Omron Sysmac Studio project comunicacion de PLC (Sysmac Studio 1.23.0.14, StandardProject)

# Controller NX1_2: NX1P2-1040DT1 version 1.18
Task PrimaryTask (priority 4, period or condition 2000): Programa0

VAR_GLOBAL
    HMI_CAMBIO_MOTORES AT %W1.0 : BOOL;  (* published *)
    HMI_MOTOR_ENCENDIDO AT %W1.2 : BOOL;  (* published *)
    hmi_pulsador_marcha1 AT %W0.00 : BOOL;  (* published *)
    hmi_pulsador_paro1 AT %W0.02 : BOOL;  (* published *)
    hmi_pulsador_inversion1 AT %W0.04 : BOOL;  (* published *)
    adelante : BOOL;  (* at BuiltInIO://cpu/#0/Output_Bit_00; network input *)
    hmi_velocidades_motor1 AT %W0.14 : BOOL;  (* published *)
    hmi_velocidades_motor2 AT %W0.12 : BOOL;  (* published *)
END_VAR
VAR_GLOBAL RETAIN
    hz_motor1_hmi AT %D6 : INT;  (* published *)
    hz_motor2_hmi AT %D4 : INT;  (* published *)
END_VAR
VAR_GLOBAL
    velocidades_motor1 : BOOL;  (* network output *)
    velocidades_motor2 : BOOL;  (* network input *)
    hz_motor1_envio : INT;  (* network input *)
    hz_motor2_envio : INT;  (* network output *)
    atras : BOOL;  (* at BuiltInIO://cpu/#0/Output_Bit_01 *)
    v1 : BOOL;  (* at BuiltInIO://cpu/#0/Output_Bit_02 *)
    v2 : BOOL;  (* at BuiltInIO://cpu/#0/Output_Bit_03 *)
    pulsador_marcha2 AT %W0.06 : BOOL;  (* published *)
    pulsador_paro2 AT %W0.08 : BOOL;  (* published *)
    pulsador_inversion2 AT %W0.10 : BOOL;  (* published *)
    NX1_2_PM_HMI_MOTOR2 : BOOL;  (* network input *)
    NX1_2_PP_HMI_MOTOR2 : BOOL;  (* network input *)
    NX1_2_INVERTIR_HMI_MOTOR2 : BOOL;  (* network input *)
    NX1_2_MOTOR2_ADELANTE : BOOL;  (* network input *)
    NX1_2_MOTOR2_ATRAS : BOOL;  (* network input *)
    NX1_2_PM_HMI_MOTOR1 : BOOL;  (* network output *)
    NX1_2_PP_HMI_MOTOR1 : BOOL;  (* network output *)
    NX1_2_INVERTIR_HMI_MOTOR1 : BOOL;  (* network output *)
    NX1_2_MOTOR1_ADELANTE : BOOL;  (* network output *)
    NX1_2_MOTOR1_ATRAS : BOOL;  (* network output *)
    marcha2 : BOOL;  (* at BuiltInIO://cpu/#0/Input_Bit_00 *)
    paro2 : BOOL;  (* at BuiltInIO://cpu/#0/Input_Bit_01 *)
    invertir2 : BOOL;  (* at BuiltInIO://cpu/#0/Input_Bit_02 *)
END_VAR

PROGRAM Programa0
VAR
    velocidadmotor2 : INT;
    sentido_telerruptor : BOOL;
    variableinversion : BOOL;
    PARO_BOTONERA : BOOL;
    PARO : BOOL;
END_VAR
VAR_EXTERNAL
    adelante : BOOL;
    atras : BOOL;
    hmi_pulsador_marcha1 : BOOL;
    NX1_2_PM_HMI_MOTOR2 : BOOL;
    hmi_pulsador_paro1 : BOOL;
    NX1_2_PP_HMI_MOTOR2 : BOOL;
    hmi_pulsador_inversion1 : BOOL;
    NX1_2_INVERTIR_HMI_MOTOR2 : BOOL;
    v1 : BOOL;
    v2 : BOOL;
    hmi_velocidades_motor2 : BOOL;
    velocidades_motor1 : BOOL;
    hmi_velocidades_motor1 : BOOL;
    velocidades_motor2 : BOOL;
    pulsador_marcha2 : BOOL;
    NX1_2_PM_HMI_MOTOR1 : BOOL;
    pulsador_paro2 : BOOL;
    NX1_2_PP_HMI_MOTOR1 : BOOL;
    NX1_2_INVERTIR_HMI_MOTOR1 : BOOL;
    pulsador_inversion2 : BOOL;
    hz_motor2_envio : INT;
    hz_motor1_envio : INT;
    hz_motor2_hmi : INT;
    hz_motor1_hmi : INT;
    invertir2 : BOOL;
    marcha2 : BOOL;
    paro2 : BOOL;
    HMI_CAMBIO_MOTORES : BOOL;
    HMI_MOTOR_ENCENDIDO : BOOL;
END_VAR
VAR
    _p1 : BOOL;
    _e2 : R_TRIG;
    _e3 : R_TRIG;
    _e4 : R_TRIG;
END_VAR

(* Section Sección0: ladder, written here as Structured Text *)

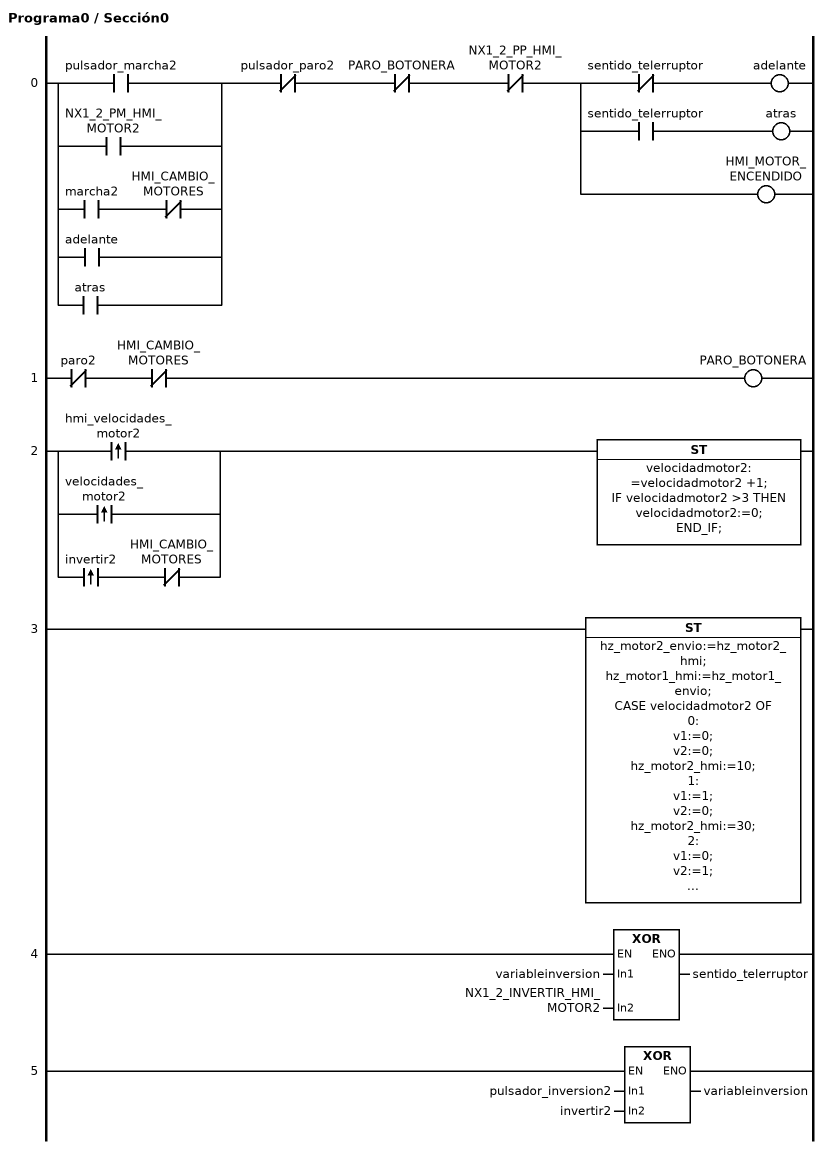
(* Rung 0 *)
_p1 := (pulsador_marcha2 OR NX1_2_PM_HMI_MOTOR2 OR (marcha2 AND NOT HMI_CAMBIO_MOTORES) OR adelante OR atras) AND NOT pulsador_paro2 AND NOT PARO_BOTONERA AND NOT NX1_2_PP_HMI_MOTOR2;
adelante := _p1 AND NOT sentido_telerruptor;
atras := _p1 AND sentido_telerruptor;
HMI_MOTOR_ENCENDIDO := _p1;
(* Rung 1 *)
PARO_BOTONERA := NOT paro2 AND NOT HMI_CAMBIO_MOTORES;
(* Rung 2 *)
_e2(CLK := hmi_velocidades_motor2);
_e3(CLK := velocidades_motor2);
_e4(CLK := invertir2);
IF _e2.Q OR _e3.Q OR (_e4.Q AND NOT HMI_CAMBIO_MOTORES) THEN
    velocidadmotor2:=velocidadmotor2 +1;
    IF velocidadmotor2 >3 THEN
    	velocidadmotor2:=0;
    END_IF;
END_IF;
(* Rung 3 *)
hz_motor2_envio:=hz_motor2_hmi;

hz_motor1_hmi:=hz_motor1_envio;

CASE velocidadmotor2 OF 
	0:
	v1:=0;
	v2:=0;
	hz_motor2_hmi:=10;
	1:
	v1:=1;
	v2:=0;
	hz_motor2_hmi:=30;
	2:
	v1:=0;
	v2:=1;
	hz_motor2_hmi:=50;
	3:
	v1:=1;
	v2:=1;
	hz_motor2_hmi:=80;
END_CASE;



	
(* Rung 4 *)
sentido_telerruptor := variableinversion XOR NX1_2_INVERTIR_HMI_MOTOR2;
(* Rung 5 *)
variableinversion := pulsador_inversion2 XOR invertir2;

(* Section Sección1: ladder, written here as Structured Text *)

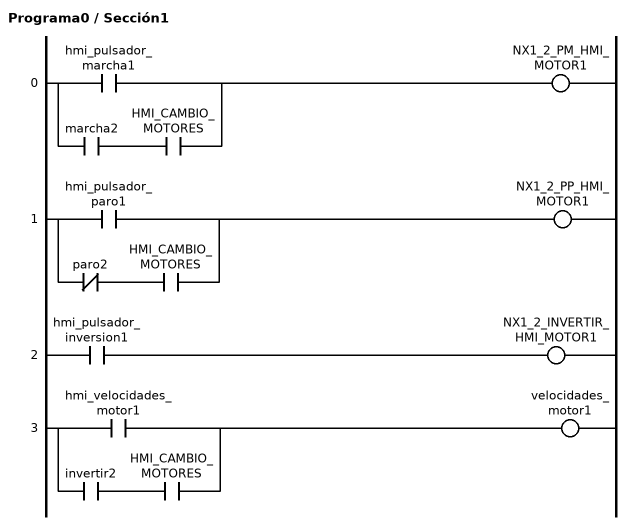
(* Rung 0 *)
NX1_2_PM_HMI_MOTOR1 := hmi_pulsador_marcha1 OR (marcha2 AND HMI_CAMBIO_MOTORES);
(* Rung 1 *)
NX1_2_PP_HMI_MOTOR1 := hmi_pulsador_paro1 OR (NOT paro2 AND HMI_CAMBIO_MOTORES);
(* Rung 2 *)
NX1_2_INVERTIR_HMI_MOTOR1 := hmi_pulsador_inversion1;
(* Rung 3 *)
velocidades_motor1 := hmi_velocidades_motor1 OR (invertir2 AND HMI_CAMBIO_MOTORES);
END_PROGRAM

# Controller NX1_1: NX1P2-1040DT1 version 1.18
Task PrimaryTask (priority 4, period or condition 2000): Programa0

VAR_GLOBAL
    NX1_1_Velocidades_Motor2 : BOOL;  (* network output *)
    NX1_1_Velocidades_Motor1 : BOOL;  (* network input *)
    Velocidades_Motor2_HMI AT %W0.12 : BOOL;  (* published *)
    Velocidades_Motor1_HMI AT %W0.14 : BOOL;  (* published *)
END_VAR
VAR_GLOBAL RETAIN
    Hz_Motor2_HMI AT %D2 : INT;  (* published *)
    Hz_Motor1_HMI AT %D6 : INT;  (* published *)
END_VAR
VAR_GLOBAL
    NX1_1_Hz_Motor2 : INT;  (* network input *)
    NX1_1_Hz_Motor1 : INT;  (* network output *)
    PM1_HMI AT %W0.00 : BOOL;  (* published *)
    PP1_HMI AT %W0.02 : BOOL;  (* published *)
    Invertir1_HMI AT %W0.04 : BOOL;  (* published *)
    PM2_HMI AT %W0.06 : BOOL;  (* published *)
    PP2_HMI AT %W0.08 : BOOL;  (* published *)
    Invertir2_HMI AT %W0.10 : BOOL;  (* published *)
    Motor_Adelante : BOOL;  (* at BuiltInIO://cpu/#0/Output_Bit_00 *)
    Motor_Atras : BOOL;  (* at BuiltInIO://cpu/#0/Output_Bit_01 *)
    NX1_1_PM_HMI_Motor1 : BOOL;  (* network input *)
    NX1_1_PP_HMI_Motor1 : BOOL;  (* network input *)
    NX1_1_Invertir_HMI_Motor1 : BOOL;  (* network input *)
    NX1_1_Motor1_Adelante : BOOL;  (* network input *)
    NX1_1_Motor1_Atras : BOOL;  (* network input *)
    NX1_1_PM_HMI_Motor2 : BOOL;  (* network output *)
    NX1_1_PP_HMI_Motor2 : BOOL;  (* network output *)
    NX1_1_Invertir_HMI_Motor2 : BOOL;  (* network output *)
    NX1_1_Motor2_Adelante : BOOL;  (* network output *)
    NX1_1_Motor2_Atras : BOOL;  (* network output *)
    MV1 : BOOL;  (* at BuiltInIO://cpu/#0/Output_Bit_02 *)
    MV2 : BOOL;  (* at BuiltInIO://cpu/#0/Output_Bit_03 *)
END_VAR

PROGRAM Programa0
VAR
    Sentido : BOOL;
    Velocidad_Motor1 : INT;
END_VAR
VAR_EXTERNAL
    Motor_Adelante : BOOL;
    Motor_Atras : BOOL;
    NX1_1_PM_HMI_Motor1 : BOOL;
    NX1_1_Motor1_Adelante : BOOL;
    NX1_1_Motor1_Atras : BOOL;
    NX1_1_Invertir_HMI_Motor1 : BOOL;
    NX1_1_PP_HMI_Motor1 : BOOL;
    PM1_HMI : BOOL;
    Invertir1_HMI : BOOL;
    PP1_HMI : BOOL;
    PM2_HMI : BOOL;
    NX1_1_Motor2_Adelante : BOOL;
    NX1_1_Motor2_Atras : BOOL;
    PP2_HMI : BOOL;
    Invertir2_HMI : BOOL;
    NX1_1_PM_HMI_Motor2 : BOOL;
    NX1_1_PP_HMI_Motor2 : BOOL;
    NX1_1_Invertir_HMI_Motor2 : BOOL;
    Velocidades_Motor1_HMI : BOOL;
    MV1 : BOOL;
    MV2 : BOOL;
    Velocidades_Motor2_HMI : BOOL;
    NX1_1_Velocidades_Motor1 : BOOL;
    NX1_1_Velocidades_Motor2 : BOOL;
    Hz_Motor1_HMI : INT;
    NX1_1_Hz_Motor1 : INT;
    NX1_1_Hz_Motor2 : INT;
    Hz_Motor2_HMI : INT;
END_VAR
VAR
    _p1 : BOOL;
    _e2 : R_TRIG;
    _e3 : R_TRIG;
END_VAR

(* Section Sección0: ladder, written here as Structured Text *)

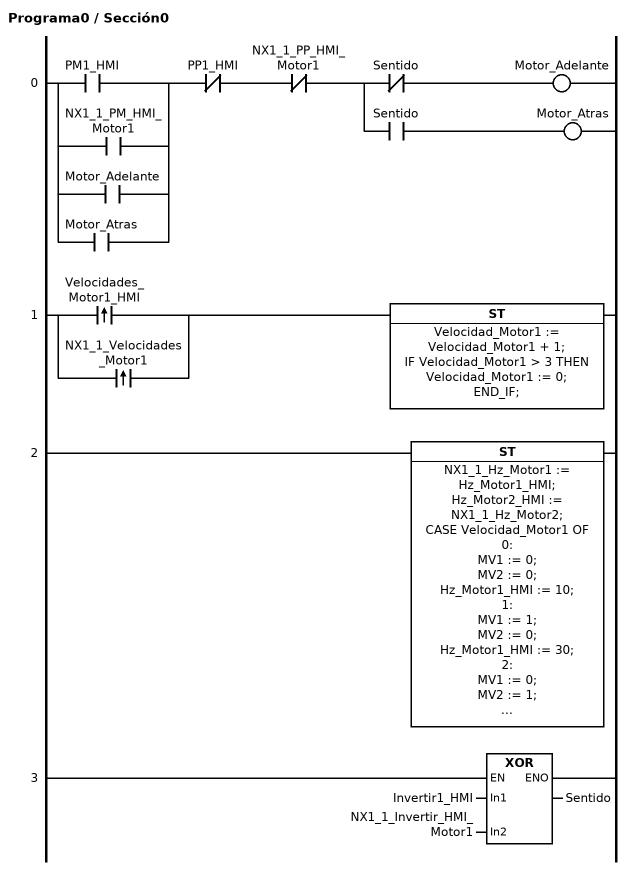
(* Rung 0 *)
_p1 := (PM1_HMI OR NX1_1_PM_HMI_Motor1 OR Motor_Adelante OR Motor_Atras) AND NOT PP1_HMI AND NOT NX1_1_PP_HMI_Motor1;
Motor_Adelante := _p1 AND NOT Sentido;
Motor_Atras := _p1 AND Sentido;
(* Rung 1 *)
_e2(CLK := Velocidades_Motor1_HMI);
_e3(CLK := NX1_1_Velocidades_Motor1);
IF _e2.Q OR _e3.Q THEN
    Velocidad_Motor1 := Velocidad_Motor1 + 1;
    IF Velocidad_Motor1 > 3 THEN
    	Velocidad_Motor1 := 0;
    END_IF;
END_IF;
(* Rung 2 *)
NX1_1_Hz_Motor1 := Hz_Motor1_HMI;
Hz_Motor2_HMI := NX1_1_Hz_Motor2;

CASE Velocidad_Motor1 OF
    0:
	MV1 := 0;
	MV2 := 0;
	Hz_Motor1_HMI := 10;
	1:
	MV1 := 1;
	MV2 := 0;
	Hz_Motor1_HMI := 30;
	2:
	MV1 := 0;
	MV2 := 1;
	Hz_Motor1_HMI := 50;
	3:
	MV1 := 1;
	MV2 := 1;
	Hz_Motor1_HMI := 80;
END_CASE;
(* Rung 3 *)
Sentido := Invertir1_HMI XOR NX1_1_Invertir_HMI_Motor1;

(* Section Sección1: ladder, written here as Structured Text *)

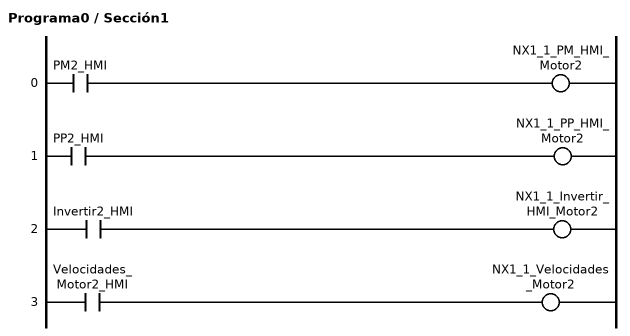
(* Rung 0 *)
NX1_1_PM_HMI_Motor2 := PM2_HMI;
(* Rung 1 *)
NX1_1_PP_HMI_Motor2 := PP2_HMI;
(* Rung 2 *)
NX1_1_Invertir_HMI_Motor2 := Invertir2_HMI;
(* Rung 3 *)
NX1_1_Velocidades_Motor2 := Velocidades_Motor2_HMI;
END_PROGRAM